FUNCTION_BLOCK FB_Read
//Permet de lire les Valeurs de max 1 semaine de points (1 pt/min pdt 7 jours)

VAR_INPUT
	InDirectory 				: T_MaxString;		// Base file of the Historization 
	InExecute					: BOOL;			//Rising Edge detection of read
END_VAR                 		

VAR_OUTPUT              		
	OutValue					: T_MaxString;
	OutCompleted				: BOOL;
	OutbBusy					: BOOL;
	OutError 					: BOOL;
	OutErrorID 					: UINT; // 1 : File not found

END_VAR                 		
VAR     
	// Initialisation 
	RS_Busy						: RS;
	Trig_Start 					: R_TRIG;
	FullDirectory				: STRING;  
	
	OpenFile					: FB_FileOpen;
	ReadFile					: FB_FileRead;
	CloseFile					: FB_FileClose;
	
	Opening						: BOOL := TRUE;
	Reading						: BOOL;
	Closing						: BOOL;
	
	EOF_Reached					: BOOL;
	
	FileHandle					: UINT;
	FileHandle_Old				: UINT;
	
	NbJours						: UINT;
	KK: UINT 					:= 1;
END_VAR

Trig_Start(CLK := InExecute);

IF Trig_Start.Q THEN 
	Outerror:= FALSE ; // On reinitialize l'error à un nouvel essai . 
	OpenFile(bExecute:= FALSE  ); 
END_IF

RS_Busy(Set := Trig_Start.Q, RESET1 := Outerror OR OutCompleted);
OutbBusy := RS_Busy.Q1;
OutCompleted := FALSE;


IF RS_Busy.Q1 THEN	
		//Ouverture du Fichier, récupération du handle
		OpenFile
		(
			sNetId := '',
			sPathName := InDirectory,
			nMode := FOPEN_MODEREAD,
			ePath := PATH_GENERIC,
			bExecute := TRUE,
			hFile => FileHandle
		);
		
		IF NOT OpenFile.bBusy AND OpenFile.bError AND OpenFile.nErrId = 1804 THEN // Le fichier n'existe pas 
			OutErrorID := 1;
			OutError := OpenFile.bError;
		ELSIF OpenFile.bError THEN		// Il y a eu une autre erreur
			OutError := OpenFile.bError;
		ELSIF NOT OpenFile.bError AND NOT OpenFile.bBusy AND FileHandle <> 0 THEN
			opening := FALSE;
		END_IF
		
		
		
		IF NOT opening AND NOT EOF_Reached THEN			
			ReadFile
			(
				sNetId := '',
				hFile := FileHandle,
				bExecute := TRUE,
				tTimeout := T#1S,
				pReadBuff := ADR(OutValue),
				cbReadLen := SIZEOF(OutValue),				
				bEOF => EOF_Reached
			);	
			IF NOT ReadFile.bBusy AND ReadFile.bError THEN
				OutError := TRUE;	
				ReadFile(bExecute := FALSE);
			ELSIF NOT ReadFile.bBusy THEN
				ReadFile(bExecute := FALSE);	
			END_IF
		ELSIF EOF_Reached THEN
			ReadFile(bExecute := FALSE);
	
			CloseFile
			(
				sNetId := '',
				bExecute := TRUE,
				hFile := FileHandle,
				tTimeout := T#1S
			);
			IF NOT CloseFile.bBusy AND NOT CloseFile.bError  THEN
				Opening := TRUE;
				EOF_Reached := FALSE;
				OpenFile(bExecute := FALSE);
				ReadFile(bExecute := FALSE);
				CloseFile(bExecute := FALSE);
				
				OUTCompleted := TRUE;
			ELSIF CloseFile.bError THEN
				OutError := TRUE;
				OutErrorID := UDINT_TO_UINT(Closefile.nErrId);
			END_IF	
		END_IF
	END_IF

END_FUNCTION_BLOCK

(* stored: Version 1.1.0.1, ProductVersion 3.1.4024.6
   POU FB_Read: Id {3734db36-5f30-4e42-af53-00437168a2f5}, SpecialFunc None *)
